(* Logix 5000 project; controller AplicacionAFEbancoDePruebas vendor 1 type 14 code 149 rev 33.12; software revision 33.01 *)

TASK MainTask (continuous, watchdog 500 ms) : MainProgram

MODULES
   Local : vendor 1 type 14 code 149 (Compact 0, rev 33.12)
      Discrete_IO : Embedded (Compact 1, rev 3.1, Output RPI 20 ms)
      PLC : 1769-L32E Ethernet Port (Ethernet 192.168.2.131, rev 20.1)
         PLC_Controller : vendor 1 type 14 code 77 (CompactLogixL32EController 0, rev 20.1, $23548359$ RPI 20 ms)
      VSD_AFE : vendor 1 type 143 code 8336 (Ethernet 192.168.2.50, rev 6.5, Output RPI 20 ms)
          : vendor 1 type 143 code 416 (RhinoBP 4, rev 1.8)
          : vendor 1 type 143 code 416 (RhinoBP 5, rev 1.8)
          : vendor 1 type 143 code 161 (RhinoBP 10, rev 1.1)
          : vendor 1 type 143 code 4770 (RhinoBP 12, rev 1.1)
          : vendor 1 type 143 code 675 (RhinoBP 13, rev 1.1)
          : vendor 1 type 143 code 2724 (RhinoBP 14, rev 1.1)
END_MODULES

VAR_GLOBAL   (* controller tags *)
   SRP_SimActualStroke : DINT;   // Variable Simulación de PLC Variador DC
END_VAR

PROGRAM MainProgram   (* main routine MainRoutine *)

ROUTINE dinagramaPotencia   (* ladder *)
END_ROUTINE

ROUTINE MainRoutine   (* ladder *)
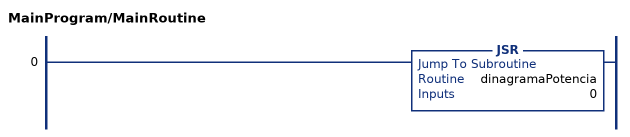
   0 (stored rung type 13): JSR(dinagramaPotencia,0);
END_ROUTINE
END_PROGRAM
